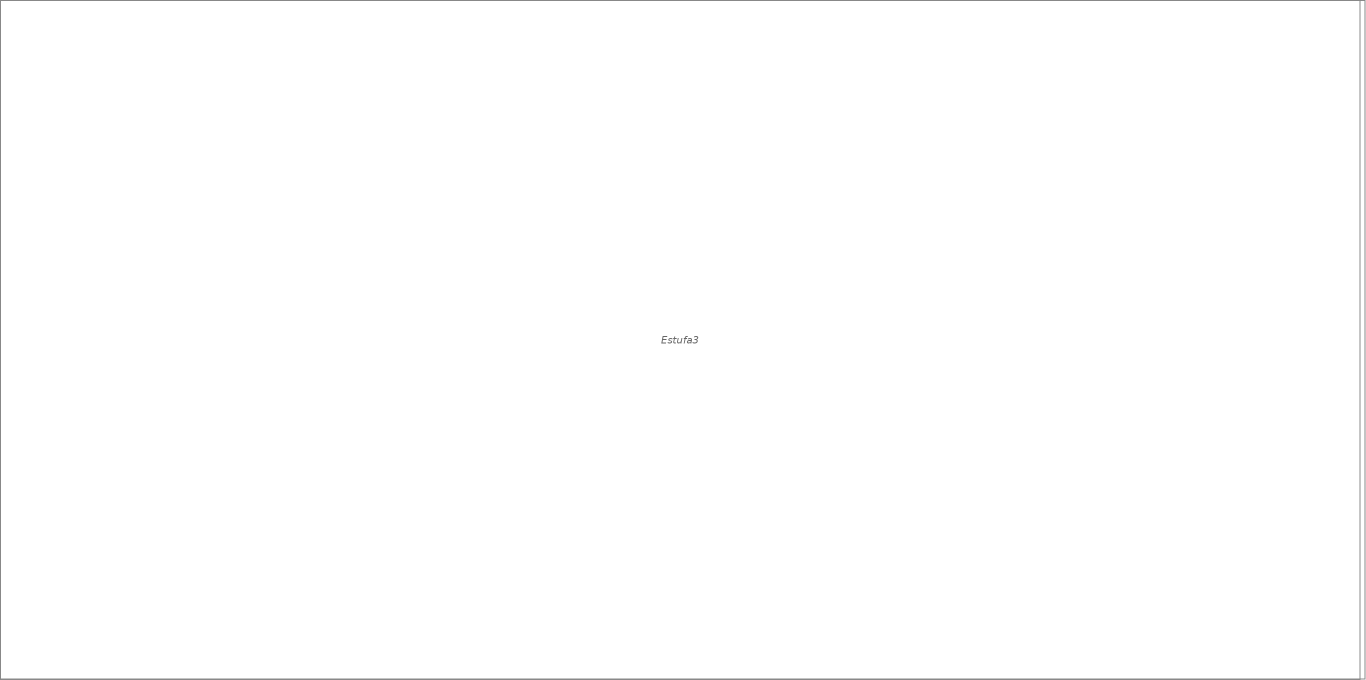
VISUALIZATION Aba_Estufa_3  // 1366x680
    TabControl (0,0 1360x680)
        shows Estufa3()
        shows Grafico_3()
        [0]: TabTitle=Dashboard
        [1]: TabTitle=Gráfico
END_VISUALIZATION

(* stored: Version 1.1.0.1, ProductVersion 3.1.4024.12
   Visu Aba_Estufa_3: Id {29fab33f-9444-496e-b8c2-795729da3958} *)
